{attribute 'qualified_only'}
{attribute 'strict'}
TYPE E_PneumaticAxisMode :
(   
	eMonostable := 0, //One stable point, single solenoid
	eBistable := 1 //Two stable points, double solenoid
):= eMonostable;
END_TYPE

(* stored: Version 1.1.0.1
   DUT E_PneumaticAxisMode: Id {8d59e371-0acf-0583-34a1-fd0fac831808} *)
